FUNCTION_BLOCK FB_TimeBasedIntegrator
VAR_INPUT
	tBaseTime:TIME:=T#1S;
	rIn:LREAL;
	addNegativeValues:BOOL;
	reset:BOOL;
END_VAR
VAR_OUTPUT
	bErr: BOOL;
END_VAR
VAR
	t1:TON;
END_VAR
VAR_IN_OUT
	rAccumulator:LREAL;
END_VAR

IF tBaseTime = T#0S THEN
	RETURN;
END_IF

t1(IN:= NOT t1.Q, PT:= tBaseTime);

IF t1.Q AND addNegativeValues THEN
	rAccumulator:=rAccumulator+rIn;
ELSIF t1.Q AND NOT addNegativeValues THEN
	rAccumulator := SEL(rIn >0, rAccumulator, rAccumulator+rIn);
END_IF

IF reset THEN
	rAccumulator:=0;
END_IF

END_FUNCTION_BLOCK

(* stored: Version 1.1.0.1, ProductVersion 3.1.4024.12
   POU FB_TimeBasedIntegrator: Id {b809bf77-0074-44c0-a221-7968b0e1dd12}, SpecialFunc None *)
